// TIA Portal V19 export
FUNCTION "A0303_Sostegno_Coda_CALL" : Void   // FC150, LAD
// stored: SetENOAutomatically false
   VAR_TEMP
      V1_Work_1 : Bool;
      V1_Work_2 : Bool;
      V1_Rest : Bool;
      V1_Rest_2 : Bool;
      V2_Work : Bool;
      V2_Rest_1 : Bool;
      V2_Rest_2 : Bool;
   END_VAR
   VAR CONSTANT
      MISSING : Int;
   END_VAR
BEGIN

REGION Network 1: DataIn - Asse Y
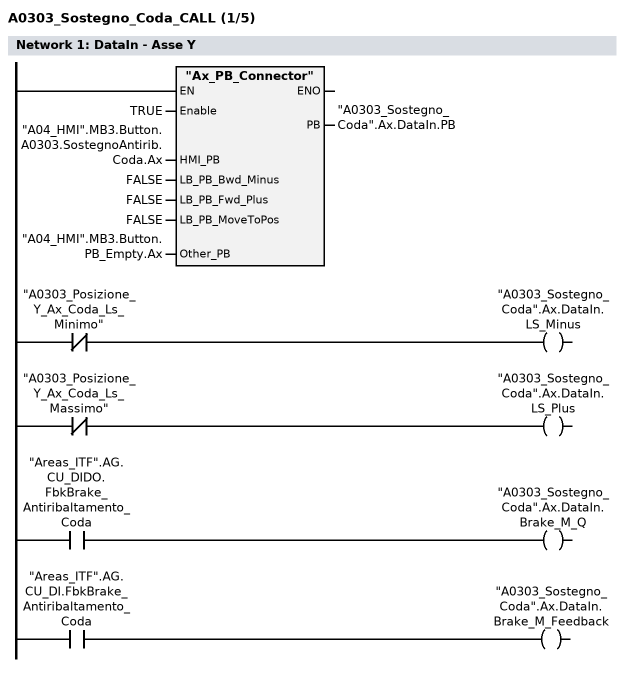
   RUNG wire#powerrail
      "Ax_PB_Connector"(Enable := TRUE, HMI_PB := "A04_HMI".MB3.Button.A0303.SostegnoAntirib.Coda.Ax, LB_PB_Bwd_Minus := FALSE, LB_PB_Fwd_Plus := FALSE, LB_PB_MoveToPos := FALSE, Other_PB := "A04_HMI".MB3.Button.PB_Empty.Ax, PB => "A0303_Sostegno_Coda".Ax.DataIn.PB)
   END_RUNG
   RUNG wire#powerrail
      I_Contact( "A0303_Posizione_Y_Ax_Coda_Ls_Minimo" )
      Coil( "A0303_Sostegno_Coda".Ax.DataIn.LS_Minus )
   END_RUNG
   RUNG wire#powerrail
      I_Contact( "A0303_Posizione_Y_Ax_Coda_Ls_Massimo" )
      Coil( "A0303_Sostegno_Coda".Ax.DataIn.LS_Plus )
   END_RUNG
   RUNG wire#powerrail
      Contact( "Areas_ITF".AG.CU_DIDO.FbkBrake_Antiribaltamento_Coda )
      Coil( "A0303_Sostegno_Coda".Ax.DataIn.Brake_M_Q )
   END_RUNG
   RUNG wire#powerrail
      Contact( "Areas_ITF".AG.CU_DI.FbkBrake_Antiribaltamento_Coda )
      Coil( "A0303_Sostegno_Coda".Ax.DataIn.Brake_M_Feedback )
   END_RUNG
   // the same network as SCL:
   "Ax_PB_Connector"(Enable := TRUE,
                     HMI_PB := "A04_HMI".MB3.Button.A0303.SostegnoAntirib.Coda.Ax,
                     LB_PB_Bwd_Minus := FALSE,
                     LB_PB_Fwd_Plus := FALSE,
                     LB_PB_MoveToPos := FALSE,
                     Other_PB := "A04_HMI".MB3.Button.PB_Empty.Ax,
                     PB => "A0303_Sostegno_Coda".Ax.DataIn.PB);
   "A0303_Sostegno_Coda".Ax.DataIn.LS_Minus := NOT "A0303_Posizione_Y_Ax_Coda_Ls_Minimo";
   "A0303_Sostegno_Coda".Ax.DataIn.LS_Plus := NOT "A0303_Posizione_Y_Ax_Coda_Ls_Massimo";
   "A0303_Sostegno_Coda".Ax.DataIn.Brake_M_Q := "Areas_ITF".AG.CU_DIDO.FbkBrake_Antiribaltamento_Coda;
   "A0303_Sostegno_Coda".Ax.DataIn.Brake_M_Feedback := "Areas_ITF".AG.CU_DI.FbkBrake_Antiribaltamento_Coda;
END_REGION

REGION Network 2: DataIn - Valve
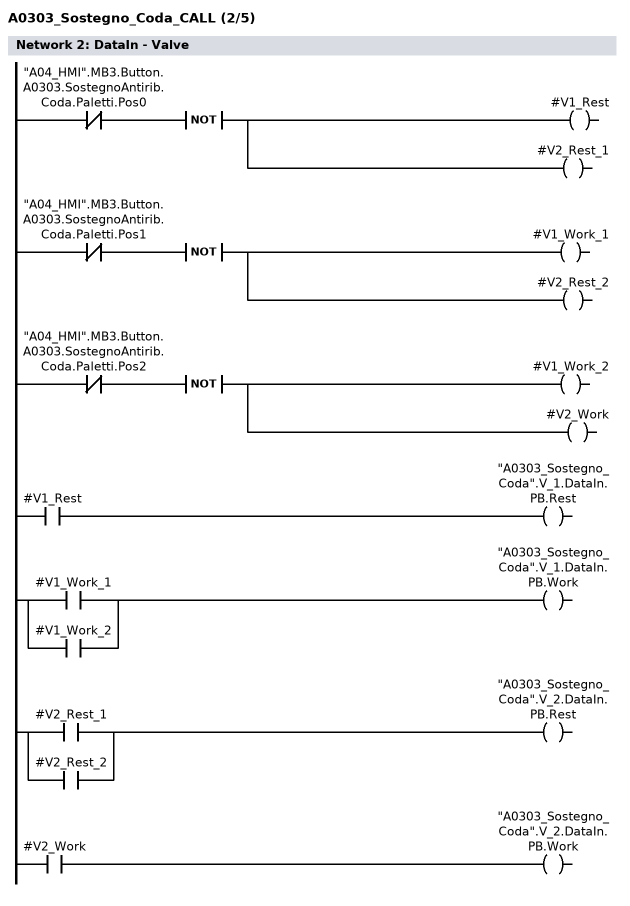
   RUNG wire#powerrail
      I_Contact( "A04_HMI".MB3.Button.A0303.SostegnoAntirib.Coda.Paletti.Pos0 )
      Not()
      wire#w1
      Coil( #V1_Rest )
   END_RUNG
   RUNG wire#w1
      Coil( #V2_Rest_1 )
   END_RUNG
   RUNG wire#powerrail
      I_Contact( "A04_HMI".MB3.Button.A0303.SostegnoAntirib.Coda.Paletti.Pos1 )
      Not()
      wire#w2
      Coil( #V1_Work_1 )
   END_RUNG
   RUNG wire#w2
      Coil( #V2_Rest_2 )
   END_RUNG
   RUNG wire#powerrail
      I_Contact( "A04_HMI".MB3.Button.A0303.SostegnoAntirib.Coda.Paletti.Pos2 )
      Not()
      wire#w3
      Coil( #V1_Work_2 )
   END_RUNG
   RUNG wire#w3
      Coil( #V2_Work )
   END_RUNG
   RUNG wire#powerrail
      Contact( #V1_Rest )
      Coil( "A0303_Sostegno_Coda".V_1.DataIn.PB.Rest )
   END_RUNG
   RUNG wire#powerrail
      Contact( #V1_Work_1 )
      wire#w4
      Coil( "A0303_Sostegno_Coda".V_1.DataIn.PB.Work )
   END_RUNG
   RUNG wire#powerrail
      Contact( #V1_Work_2 )
   END_RUNG wire#w4
   RUNG wire#powerrail
      Contact( #V2_Rest_1 )
      wire#w5
      Coil( "A0303_Sostegno_Coda".V_2.DataIn.PB.Rest )
   END_RUNG
   RUNG wire#powerrail
      Contact( #V2_Rest_2 )
   END_RUNG wire#w5
   RUNG wire#powerrail
      Contact( #V2_Work )
      Coil( "A0303_Sostegno_Coda".V_2.DataIn.PB.Work )
   END_RUNG
   // the same network as SCL:
   #V1_Rest := NOT (NOT "A04_HMI".MB3.Button.A0303.SostegnoAntirib.Coda.Paletti.Pos0);
   #V2_Rest_1 := NOT (NOT "A04_HMI".MB3.Button.A0303.SostegnoAntirib.Coda.Paletti.Pos0);
   #V1_Work_1 := NOT (NOT "A04_HMI".MB3.Button.A0303.SostegnoAntirib.Coda.Paletti.Pos1);
   #V2_Rest_2 := NOT (NOT "A04_HMI".MB3.Button.A0303.SostegnoAntirib.Coda.Paletti.Pos1);
   #V1_Work_2 := NOT (NOT "A04_HMI".MB3.Button.A0303.SostegnoAntirib.Coda.Paletti.Pos2);
   #V2_Work := NOT (NOT "A04_HMI".MB3.Button.A0303.SostegnoAntirib.Coda.Paletti.Pos2);
   "A0303_Sostegno_Coda".V_1.DataIn.PB.Rest := #V1_Rest;
   "A0303_Sostegno_Coda".V_1.DataIn.PB.Work := #V1_Work_1 OR #V1_Work_2;
   "A0303_Sostegno_Coda".V_2.DataIn.PB.Rest := #V2_Rest_1 OR #V2_Rest_2;
   "A0303_Sostegno_Coda".V_2.DataIn.PB.Work := #V2_Work;
END_REGION

REGION Network 3: DataIn - Valve
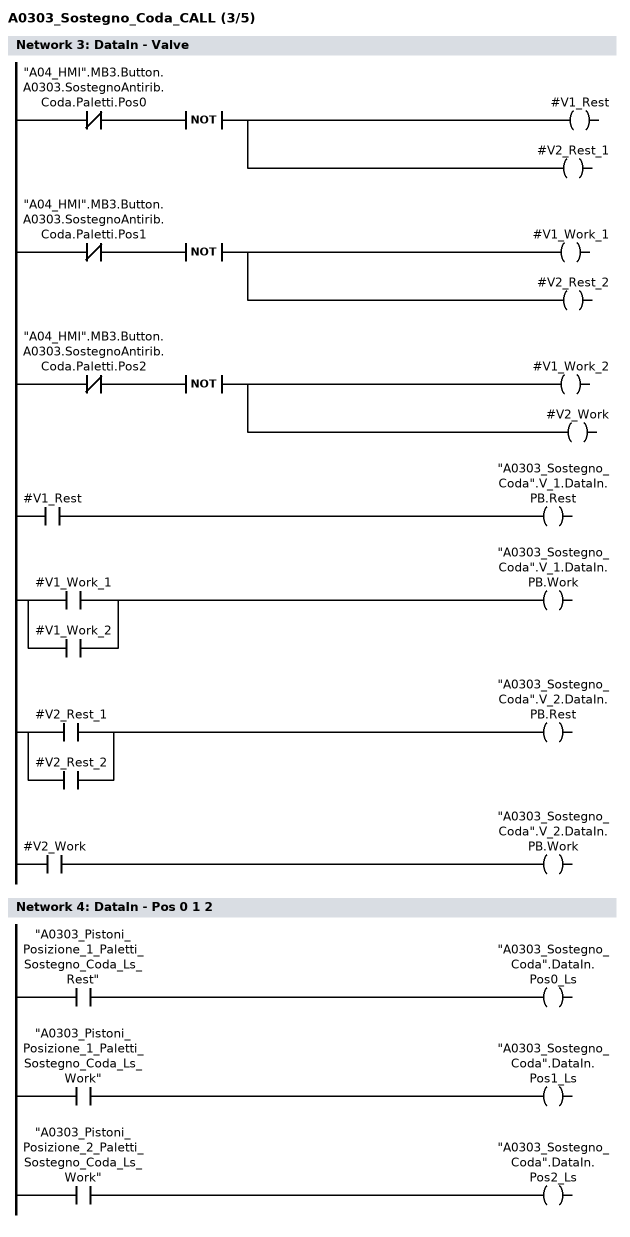
   RUNG wire#powerrail
      I_Contact( "A04_HMI".MB3.Button.A0303.SostegnoAntirib.Coda.Paletti.Pos0 )
      Not()
      wire#w1
      Coil( #V1_Rest )
   END_RUNG
   RUNG wire#w1
      Coil( #V2_Rest_1 )
   END_RUNG
   RUNG wire#powerrail
      I_Contact( "A04_HMI".MB3.Button.A0303.SostegnoAntirib.Coda.Paletti.Pos1 )
      Not()
      wire#w2
      Coil( #V1_Work_1 )
   END_RUNG
   RUNG wire#w2
      Coil( #V2_Rest_2 )
   END_RUNG
   RUNG wire#powerrail
      I_Contact( "A04_HMI".MB3.Button.A0303.SostegnoAntirib.Coda.Paletti.Pos2 )
      Not()
      wire#w3
      Coil( #V1_Work_2 )
   END_RUNG
   RUNG wire#w3
      Coil( #V2_Work )
   END_RUNG
   RUNG wire#powerrail
      Contact( #V1_Rest )
      Coil( "A0303_Sostegno_Coda".V_1.DataIn.PB.Rest )
   END_RUNG
   RUNG wire#powerrail
      Contact( #V1_Work_1 )
      wire#w4
      Coil( "A0303_Sostegno_Coda".V_1.DataIn.PB.Work )
   END_RUNG
   RUNG wire#powerrail
      Contact( #V1_Work_2 )
   END_RUNG wire#w4
   RUNG wire#powerrail
      Contact( #V2_Rest_1 )
      wire#w5
      Coil( "A0303_Sostegno_Coda".V_2.DataIn.PB.Rest )
   END_RUNG
   RUNG wire#powerrail
      Contact( #V2_Rest_2 )
   END_RUNG wire#w5
   RUNG wire#powerrail
      Contact( #V2_Work )
      Coil( "A0303_Sostegno_Coda".V_2.DataIn.PB.Work )
   END_RUNG
   // the same network as SCL:
   #V1_Rest := NOT (NOT "A04_HMI".MB3.Button.A0303.SostegnoAntirib.Coda.Paletti.Pos0);
   #V2_Rest_1 := NOT (NOT "A04_HMI".MB3.Button.A0303.SostegnoAntirib.Coda.Paletti.Pos0);
   #V1_Work_1 := NOT (NOT "A04_HMI".MB3.Button.A0303.SostegnoAntirib.Coda.Paletti.Pos1);
   #V2_Rest_2 := NOT (NOT "A04_HMI".MB3.Button.A0303.SostegnoAntirib.Coda.Paletti.Pos1);
   #V1_Work_2 := NOT (NOT "A04_HMI".MB3.Button.A0303.SostegnoAntirib.Coda.Paletti.Pos2);
   #V2_Work := NOT (NOT "A04_HMI".MB3.Button.A0303.SostegnoAntirib.Coda.Paletti.Pos2);
   "A0303_Sostegno_Coda".V_1.DataIn.PB.Rest := #V1_Rest;
   "A0303_Sostegno_Coda".V_1.DataIn.PB.Work := #V1_Work_1 OR #V1_Work_2;
   "A0303_Sostegno_Coda".V_2.DataIn.PB.Rest := #V2_Rest_1 OR #V2_Rest_2;
   "A0303_Sostegno_Coda".V_2.DataIn.PB.Work := #V2_Work;
END_REGION

REGION Network 4: DataIn - Pos 0 1 2
   RUNG wire#powerrail
      Contact( "A0303_Pistoni_Posizione_1_Paletti_Sostegno_Coda_Ls_Rest" )
      Coil( "A0303_Sostegno_Coda".DataIn.Pos0_Ls )
   END_RUNG
   RUNG wire#powerrail
      Contact( "A0303_Pistoni_Posizione_1_Paletti_Sostegno_Coda_Ls_Work" )
      Coil( "A0303_Sostegno_Coda".DataIn.Pos1_Ls )
   END_RUNG
   RUNG wire#powerrail
      Contact( "A0303_Pistoni_Posizione_2_Paletti_Sostegno_Coda_Ls_Work" )
      Coil( "A0303_Sostegno_Coda".DataIn.Pos2_Ls )
   END_RUNG
   // the same network as SCL:
   "A0303_Sostegno_Coda".DataIn.Pos0_Ls := "A0303_Pistoni_Posizione_1_Paletti_Sostegno_Coda_Ls_Rest";
   "A0303_Sostegno_Coda".DataIn.Pos1_Ls := "A0303_Pistoni_Posizione_1_Paletti_Sostegno_Coda_Ls_Work";
   "A0303_Sostegno_Coda".DataIn.Pos2_Ls := "A0303_Pistoni_Posizione_2_Paletti_Sostegno_Coda_Ls_Work";
END_REGION

REGION Network 5: DataIn - OP
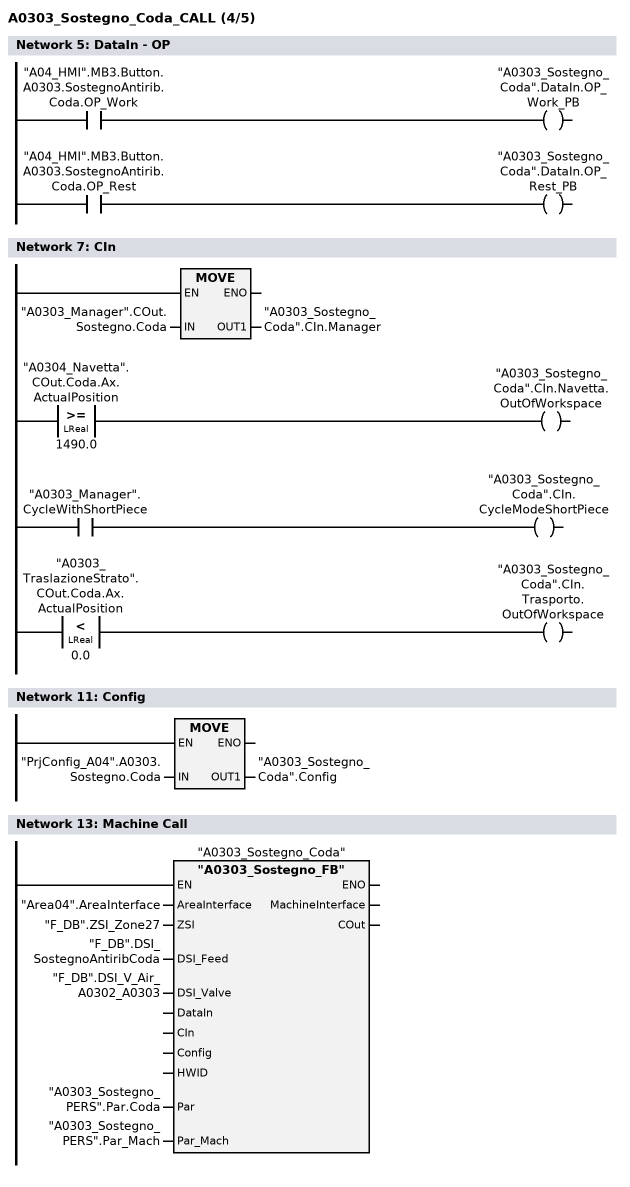
   RUNG wire#powerrail
      Contact( "A04_HMI".MB3.Button.A0303.SostegnoAntirib.Coda.OP_Work )
      Coil( "A0303_Sostegno_Coda".DataIn.OP_Work_PB )
   END_RUNG
   RUNG wire#powerrail
      Contact( "A04_HMI".MB3.Button.A0303.SostegnoAntirib.Coda.OP_Rest )
      Coil( "A0303_Sostegno_Coda".DataIn.OP_Rest_PB )
   END_RUNG
   // the same network as SCL:
   "A0303_Sostegno_Coda".DataIn.OP_Work_PB := "A04_HMI".MB3.Button.A0303.SostegnoAntirib.Coda.OP_Work;
   "A0303_Sostegno_Coda".DataIn.OP_Rest_PB := "A04_HMI".MB3.Button.A0303.SostegnoAntirib.Coda.OP_Rest;
END_REGION

REGION Network 7: CIn
   RUNG wire#powerrail
      Move(in := "A0303_Manager".COut.Sostegno.Coda, out1 => "A0303_Sostegno_Coda".CIn.Manager)
   END_RUNG
   RUNG wire#powerrail
      { S7_Templates := "SrcType := LReal" } GE_Contact(in1 := "A0304_Navetta".COut.Coda.Ax.ActualPosition, in2 := 1490.0)
      Coil( "A0303_Sostegno_Coda".CIn.Navetta.OutOfWorkspace )
   END_RUNG
   RUNG wire#powerrail
      Contact( "A0303_Manager".CycleWithShortPiece )
      Coil( "A0303_Sostegno_Coda".CIn.CycleModeShortPiece )
   END_RUNG
   RUNG wire#powerrail
      { S7_Templates := "SrcType := LReal" } LT_Contact(in1 := "A0303_TraslazioneStrato".COut.Coda.Ax.ActualPosition, in2 := 0.0)
      Coil( "A0303_Sostegno_Coda".CIn.Trasporto.OutOfWorkspace )
   END_RUNG
   // the same network as SCL:
   "A0303_Sostegno_Coda".CIn.Manager := "A0303_Manager".COut.Sostegno.Coda;
   "A0303_Sostegno_Coda".CIn.Navetta.OutOfWorkspace := "A0304_Navetta".COut.Coda.Ax.ActualPosition >= 1490.0;
   "A0303_Sostegno_Coda".CIn.CycleModeShortPiece := "A0303_Manager".CycleWithShortPiece;
   "A0303_Sostegno_Coda".CIn.Trasporto.OutOfWorkspace := "A0303_TraslazioneStrato".COut.Coda.Ax.ActualPosition < 0.0;
END_REGION

REGION Network 9 (SCL): Drive
   "A0303_Sostegno_Coda".Ax.Drive.Infeed_ON := "Areas_ITF".AG.Infeed_Running;
   "A0303_Sostegno_Coda".Ax.Drive.AccessPoint := "HW_Const_Values".CU8_PN_615A1_ModuleAccessPoint;
   "A0303_Sostegno_Coda".Ax.Drive.AxisID := "CU8_ID_7_2350A1_2_2370M1";
   "A0303_Sostegno_Coda".Ax.Drive.TokenChain :="TOKENCHAIN_CU8";
END_REGION

REGION Network 10 (SCL): HW
   "A0303_Sostegno_Coda".HWID.Ax_TEL1 := "HW_Const_Values".CU8_PN_2350A1_2_Standard_telegram_1;

   "A0303_Sostegno_Coda".HWID.Enc_IO := "HW_Const_Values".HW_2374P1_Telegram_81_DI_DO;
END_REGION

REGION Network 11: Config
   RUNG wire#powerrail
      Move(in := "PrjConfig_A04".A0303.Sostegno.Coda, out1 => "A0303_Sostegno_Coda".Config)
   END_RUNG
   // the same network as SCL:
   "A0303_Sostegno_Coda".Config := "PrjConfig_A04".A0303.Sostegno.Coda;
END_REGION

REGION Network 13: Machine Call
   RUNG wire#powerrail
      "A0303_Sostegno_Coda"(AreaInterface := "Area04".AreaInterface, ZSI := "F_DB".ZSI_Zone27, DSI_Feed := "F_DB".DSI_SostegnoAntiribCoda, DSI_Valve := "F_DB".DSI_V_Air_A0302_A0303, DataIn :=, CIn :=, Config :=, HWID :=, Par := "A0303_Sostegno_PERS".Par.Coda, Par_Mach := "A0303_Sostegno_PERS".Par_Mach, MachineInterface =>, COut =>)
   END_RUNG
   // the same network as SCL:
   "A0303_Sostegno_Coda"(AreaInterface := "Area04".AreaInterface,   // "A0303_Sostegno_FB"
                         ZSI := "F_DB".ZSI_Zone27,
                         DSI_Feed := "F_DB".DSI_SostegnoAntiribCoda,
                         DSI_Valve := "F_DB".DSI_V_Air_A0302_A0303,
                         Par := "A0303_Sostegno_PERS".Par.Coda,
                         Par_Mach := "A0303_Sostegno_PERS".Par_Mach);
END_REGION

REGION Network 15: DataOut - Valve 1
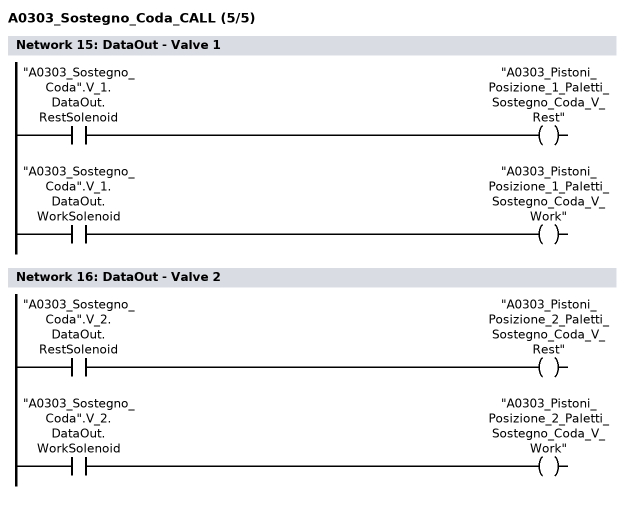
   RUNG wire#powerrail
      Contact( "A0303_Sostegno_Coda".V_1.DataOut.RestSolenoid )
      Coil( "A0303_Pistoni_Posizione_1_Paletti_Sostegno_Coda_V_Rest" )
   END_RUNG
   RUNG wire#powerrail
      Contact( "A0303_Sostegno_Coda".V_1.DataOut.WorkSolenoid )
      Coil( "A0303_Pistoni_Posizione_1_Paletti_Sostegno_Coda_V_Work" )
   END_RUNG
   // the same network as SCL:
   "A0303_Pistoni_Posizione_1_Paletti_Sostegno_Coda_V_Rest" := "A0303_Sostegno_Coda".V_1.DataOut.RestSolenoid;
   "A0303_Pistoni_Posizione_1_Paletti_Sostegno_Coda_V_Work" := "A0303_Sostegno_Coda".V_1.DataOut.WorkSolenoid;
END_REGION

REGION Network 16: DataOut - Valve 2
   RUNG wire#powerrail
      Contact( "A0303_Sostegno_Coda".V_2.DataOut.RestSolenoid )
      Coil( "A0303_Pistoni_Posizione_2_Paletti_Sostegno_Coda_V_Rest" )
   END_RUNG
   RUNG wire#powerrail
      Contact( "A0303_Sostegno_Coda".V_2.DataOut.WorkSolenoid )
      Coil( "A0303_Pistoni_Posizione_2_Paletti_Sostegno_Coda_V_Work" )
   END_RUNG
   // the same network as SCL:
   "A0303_Pistoni_Posizione_2_Paletti_Sostegno_Coda_V_Rest" := "A0303_Sostegno_Coda".V_2.DataOut.RestSolenoid;
   "A0303_Pistoni_Posizione_2_Paletti_Sostegno_Coda_V_Work" := "A0303_Sostegno_Coda".V_2.DataOut.WorkSolenoid;
END_REGION
END_FUNCTION
